FUNCTION_BLOCK CollisionGroup IMPLEMENTS ICollisionGroup
VAR_INPUT
END_VAR
VAR_OUTPUT
END_VAR
VAR
	_caGroup : Tc3_McCoordinatedMotion.AXES_GROUP_REF;
	readStatus : Tc3_McCoordinatedMotion.MC_GroupReadStatus;
	resetCAGroup : ResetGroup(THIS^);
	enableCAGroup : EnableGroup(THIS^);
	disableCAGroup : DisableGroup(this^);
END_VAR

readStatus(
	AxesGroup:= _caGroup, 
	Enable:= TRUE );
resetCAGroup();
enableCAGroup();
disableCAGroup();

METHOD Disable : BOOL
VAR_INPUT
END_VAR
IF NOT disableCAGroup.Busy THEN
	disableCAGroup.Execute();
END_IF
END_METHOD

METHOD Enable : BOOL
VAR_INPUT
END_VAR
IF NOT enableCAGroup.Busy THEN
	enableCAGroup.Execute();
END_IF
END_METHOD

PROPERTY GroupRef : reference to AXES_GROUP_REF
GET
GroupRef REF= _caGroup;
END_GET
END_PROPERTY

PROPERTY GroupState : CAGroupStatus
GET
IF readStatus.GroupDisabled THEN
	GroupState := CAGroupStatus.mcGroupStateDisabled;
ELSIF readStatus.GroupErrorStop THEN
	GroupState := CAGroupStatus.mcGroupStateErrorStop;
ELSIF readStatus.GroupHoming THEN
	GroupState := CAGroupStatus.mcGroupStateHoming;
ELSIF readStatus.GroupMoving THEN
	GroupState := CAGroupStatus.mcGroupStateMoving;
ELSIF readStatus.GroupNotReady THEN
	GroupState := CAGroupStatus.mcGroupStateNotReady;
ELSIF readStatus.GroupStandby THEN
	GroupState := CAGroupStatus.mcGroupStateStandby;
ELSIF readStatus.GroupStopping THEN
	GroupState := CAGroupStatus.mcGroupStateStopping;
ELSIF readStatus.Error THEN
	GroupState := CAGroupStatus.mcGroupError;
END_IF
END_GET
END_PROPERTY

{warning 'add method implementation '}
METHOD Reset : BOOL
IF NOT resetCAGroup.Busy THEN
	resetCAGroup.Execute();
END_IF
END_METHOD

END_FUNCTION_BLOCK

(* stored: Version 1.1.0.1, ProductVersion 3.1.4024.11
   POU CollisionGroup: Id {b63d0f8a-da32-4cf6-8258-15f9bf9b31c8}, SpecialFunc None
   Method Disable: Id {4f23215c-02ff-4fed-8568-47c96a9530ee}
   Method Enable: Id {ec0b472f-0008-427f-9be7-8c058728e9da}
   Property GroupRef: Id {fc240e72-7177-4e0d-91ed-cbdf0453df9b}
   Get Get: Id {3af383a5-c1e1-45c0-8ba8-a169a84810c4}
   Property GroupState: Id {50827d04-4f5b-4b0f-9af3-77a26ee1cb02}
   Get Get: Id {cc8632ba-7b56-4341-9258-108f345a5721}
   Method Reset: Id {14b05e09-75bc-4065-9920-b4ece711f91b} *)
